Fanuc KAREL source: compact_preamble.KL

PROGRAM KB00118
%NOLOCKGROUP
VAR
P1 : STRING[80];P2:BOOLEAN;P3:BOOLEAN
BEGIN
P1='A'
P2=TRUE
P3=TRUE
LOAD_STATUS(P1,P2,P3)
END KB00118
